SUBAPPLICATION Uebung_006a5_AX (* SR und T-Flip-Flop als Rastend/Tastend Implementierung *)
  (* Standard: 61499-2; Description: Copyright (c) 2023 Meisterschulen am Ostbahnhof This program and the accompanying materials are made available under the terms of the Eclipse Public License 2.0 which is available at https://www.eclipse.org/legal/epl-2.0/ SPDX-License-Identifier: EPL-2.0 *)
  (* Version 1.0, 2026-01-15, Franz Höpfinger, Meisterschulen am Ostbahnhof, initial API and implementation and/or initial documentation *)
  PACKAGE Uebungen;
  IMPORT logiBUS::io::DI::logiBUS_DI::Input_I1;
  IMPORT logiBUS::io::DI::logiBUS_DI_Events::BUTTON_LONG_PRESS_START;
  IMPORT logiBUS::io::DI::logiBUS_DI_Events::BUTTON_LONG_PRESS_UP;
  IMPORT logiBUS::io::DI::logiBUS_DI_Events::BUTTON_SINGLE_CLICK;
  IMPORT logiBUS::io::DQ::logiBUS_DO::Output_Q1;
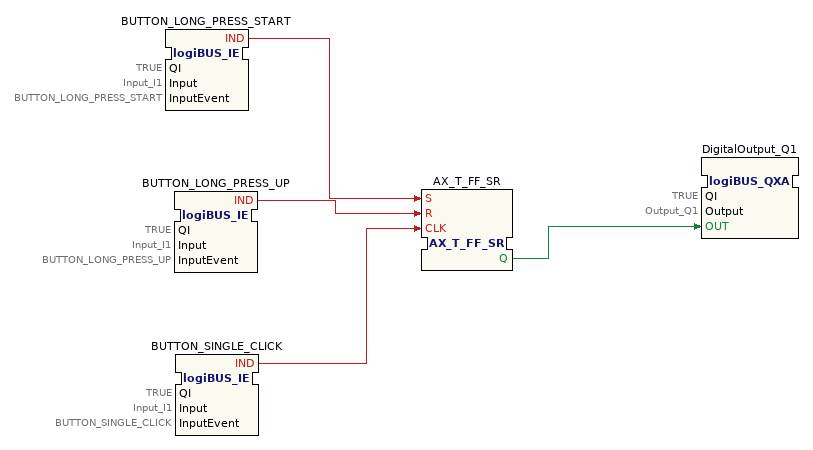
  (* Universal Eingang: so können wir mit einem Taster ODER  einem Schalter arbeiten. *)
  FBS
    BUTTON_LONG_PRESS_START : logiBUS::io::DI::logiBUS_IE(QI := TRUE, Input := Input_I1, InputEvent := BUTTON_LONG_PRESS_START);
    BUTTON_LONG_PRESS_UP : logiBUS::io::DI::logiBUS_IE(QI := TRUE, Input := Input_I1, InputEvent := BUTTON_LONG_PRESS_UP);
    AX_T_FF_SR : adapter::events::unidirectional::AX_T_FF_SR;
    BUTTON_SINGLE_CLICK : logiBUS::io::DI::logiBUS_IE(QI := TRUE, Input := Input_I1, InputEvent := BUTTON_SINGLE_CLICK);
    DigitalOutput_Q1 : logiBUS::io::DQ::logiBUS_QXA(QI := TRUE, Output := Output_Q1);
  END_FBS
  EVENT_CONNECTIONS
    BUTTON_LONG_PRESS_START.IND TO AX_T_FF_SR.S;
    BUTTON_LONG_PRESS_UP.IND TO AX_T_FF_SR.R;
    BUTTON_SINGLE_CLICK.IND TO AX_T_FF_SR.CLK;
  END_CONNECTIONS
  ADAPTER_CONNECTIONS
    AX_T_FF_SR.Q TO DigitalOutput_Q1.OUT;
  END_CONNECTIONS
END_SUBAPPLICATION
